PROGRAM Trips
VAR
	ContactDelay_TON : TON;
	ContactDelay_PT	: TIME:= T#2S;
	ContactDelay_ET	: TIME;
END_VAR

Trips_DB.CageDoorNotClose 		:= NOT MCP_IO.DoorSWclose;
Trips_DB.ChargerSummaryFault 	:= MCP_IO.Charger[1].SummaryFaulted;
Trips_DB.EStopPBpressed 		:= NOT MCP_IO.EStopPB_NotPressed;

IF (MCP_IO.ShortContactClose = TRUE AND MCP_IO.UnshortContactClose = TRUE) OR 
	(MCP_IO.ShortContactClose = FALSE AND MCP_IO.UnshortContactClose = FALSE)
	THEN
		ContactDelay_TON(IN := TRUE, PT := ContactDelay_PT, ET => ContactDelay_ET);
		ELSE
			ContactDelay_TON(IN := FALSE);
END_IF

IF ContactDelay_TON.Q = TRUE THEN 
	Trips_DB.ShortingSystemUnknown := TRUE;
	ContactDelay_TON(IN := FALSE);
END_IF

END_PROGRAM

(* stored: Version 1.1.0.1, ProductVersion 3.1.4024.11
   POU Trips: Id {8fb47083-e29f-481d-936d-668a5058e7c9}, SpecialFunc None *)
